{attribute 'linkalways'} 
{attribute 'no_explicit_call' := 'This FB is a CLASS and must be accessed using methods or properties'}
{attribute 'enable_dynamic_creation'}
FUNCTION_BLOCK _HRESULT EXTENDS DatatypeBase
VAR
	localData : HRESULT;
	activeData : REFERENCE TO HRESULT REF= localData;
END_VAR

PROPERTY PUBLIC Address : PVOID
GET
Address := ADR(activeData);
END_GET
END_PROPERTY

METHOD PUBLIC ClearReference
VAR_INPUT
END_VAR
activeData REF= localData;
END_METHOD

METHOD FB_init : BOOL
VAR_INPUT
	bInitRetains : BOOL; // if TRUE, the retain variables are initialized (warm start / cold start)
	bInCopyCode : BOOL;  // if TRUE, the instance afterwards gets moved into the copy code (online change)
	InitalValue : HRESULT;
END_VAR
localData := InitalValue;
END_METHOD

PROPERTY PUBLIC Identifier : T_MAXSTRING
GET
Identifier := 'HRESULT';
END_GET
END_PROPERTY

METHOD PUBLIC SerializeTypeWith
VAR_INPUT
	Serializer : I_Serializer;
END_VAR
Serializer.StartObject();
Serializer.AddKeyString('name','HRESULT');
Serializer.AddKeyString('type','ALIAS');
Serializer.AddKeyString('baseType','DINT');
Serializer.EndObject();
END_METHOD

METHOD PUBLIC SerializeWith
VAR_INPUT
	Serializer : I_Serializer;
END_VAR
Serializer.AddDint(activeData);
END_METHOD

PROPERTY PUBLIC Size : UDINT
GET
Size := SIZEOF(activeData);
END_GET
END_PROPERTY

METHOD TryDeserializeFrom : BOOL
VAR_INPUT
	Deserializer : I_Deserializer;
END_VAR
TryDeserializeFrom := Deserializer.TryGetDint(activeData);
END_METHOD

METHOD TryMakeReferenceOf : BOOL
VAR_INPUT
	Target : I_Datatype;
END_VAR
VAR
	pTargetData : POINTER TO HRESULT;
END_VAR
IF NOT (Target.Identifier = Identifier) THEN
	RETURN;
END_IF

pTargetData := Target.Address;
activeData REF= pTargetData^;
TryMakeReferenceOf := TRUE;
END_METHOD

PROPERTY PUBLIC Value : HRESULT
GET
Value := activeData;
END_GET
SET
activeData := Value;
END_SET
END_PROPERTY

END_FUNCTION_BLOCK

(* stored: Version 1.1.0.1, ProductVersion 3.1.4024.12
   POU _HRESULT: Id {812bad4a-7bd2-0ca8-1e32-53ad4f652147}, SpecialFunc None
   Folder Constructor: Id {c86d702f-77a8-0c2d-2692-85b706f92094}
   Property Address: Id {eaea8ce2-d780-069a-2354-b9040dbfdf59}
   Get Get: Id {9ca66335-2df6-0b97-035a-cfdc96d663e4}
   Method ClearReference: Id {3b3306cf-50f2-0e29-0162-910cb3f73574}
   Method FB_init: Id {86e1a4c2-65f3-05c8-1412-88763e434d4e}
   Property Identifier: Id {783e0e3e-7447-0c8f-3ba4-419752f4a16d}
   Get Get: Id {48ca57da-3d4d-0ccb-0db1-4ab3be926971}
   Method SerializeTypeWith: Id {79420e18-4568-0164-3ff9-5586c365a9bc}
   Method SerializeWith: Id {383560a3-8b65-0257-31d6-71c64440cf07}
   Property Size: Id {78fc7983-bbf0-072e-3bed-9c1f413ab6ff}
   Get Get: Id {1ef01c66-9a0c-0188-28d6-15ce2d32f45d}
   Method TryDeserializeFrom: Id {2cbaac55-0de2-0fcc-24d0-d8a31addeef5}
   Method TryMakeReferenceOf: Id {43bcd589-1009-0f1a-3a87-0d5bc8645b2a}
   Property Value: Id {85c486dd-d750-0c76-00cb-4c376724f1d2}
   Get Get: Id {d04c4bc3-8e0b-04d3-3b2c-700ab80225ae}
   Set Set: Id {44e9d433-2f91-0b46-3692-b60205dde3fd} *)
